PROGRAM MAIN
VAR
END_VAR

END_PROGRAM

(* stored: Version 1.1.0.1
   POU MAIN: Id {d24d79c3-2ef5-49a9-88ed-c4ba78e1268d}, SpecialFunc None *)
